// TIA Portal V21 export
VAR_GLOBAL   // PLC tag table "K_Percorsi"
END_VAR
VAR_GLOBAL CONSTANT   // user constants
   K_Percorso1 : Int := 1;
   K_Percorso2 : Int := 2;
   K_Percorso3 : Int := 3;
   K_Percorso4 : Int := 4;
   K_Percorso5 : Int := 5;
   K_Percorso6 : Int := 6;
   K_Percorso7 : Int := 7;
   K_Percorso8 : Int := 8;
   K_Percorso9 : Int := 9;
   K_Percorso10 : Int := 10;
END_VAR
